// TIA Portal V16 export
// export: Created 2021-09-08T12:44:32.1478709Z, ExportSetting WithDefaults, DisplayName Totally Integrated Automation Portal, DisplayVersion V16 Update 3, DisplayName TIA Portal Version Control Interface, DisplayVersion V16 Update 2, DisplayName TIA Portal Openness, DisplayVersion V16 Update 3, DisplayName TIA Portal Teamcenter Gateway, DisplayVersion V16, DisplayName STEP 7 Professional, DisplayVersion V16 Update 3, DisplayName STEP 7 Safety, DisplayVersion V16, DisplayName WinCC Advanced, DisplayVersion V16 Update 3
VAR_GLOBAL   // PLC tag table "A1_DQ"
   Tag_1 AT %Q0.0 : Bool;
   qP301_Start AT %Q0.1 : Bool;   // P301 Пуск
   qP302_Start AT %Q0.2 : Bool;   // P302 Пуск
   qP1201_Start AT %Q0.3 : Bool;   // P1201 Пуск
   qP1202_Start AT %Q0.4 : Bool;   // P1202 Пуск
   qP1501_Start AT %Q0.5 : Bool;   // P1501 Пуск
   qP1502_Start AT %Q0.6 : Bool;   // P1502 Пуск
   qP701_Start AT %Q0.7 : Bool;   // P701 Пуск
   qP702_Start AT %Q1.0 : Bool;   // P702 Пуск
   qP2001_Start AT %Q1.1 : Bool;   // P2001 Пуск
END_VAR
VAR_GLOBAL CONSTANT   // user constants
   iTag_1 : Int := 0;
   "qP-301_Start" : Int := 1;
   "qP-302_Start" : Int := 2;
   "qP-1201_Start" : Int := 3;
   "qP-1202_Start" : Int := 4;
   "qP-1501_Start" : Int := 5;
   "qP-1502_Start" : Int := 6;
   "qP-701_Start" : Int := 7;
   "qP-702_Start" : Int := 8;
   "qP-2001_Start" : Int := 9;
END_VAR
